(*******************************************************************************
                          protoc-gen-twincat V0.0.0.0                           
             https://github.bhs-world.com/CorrML/protoc-gen-twincat             
*******************************************************************************)
{attribute 'no_explicit_call' := 'do not call this POU directly'}
{attribute 'no-analysis'}
FUNCTION_BLOCK INTERNAL FINAL FB_Baz IMPLEMENTS I_Message
VAR
    _fbMessageParser : FB_MessageParser(ipMessage:= THIS^);
    _fbMessageWriter : FB_MessageWriter(ipMessage:= THIS^);
    _stBaz : ST_Baz;
    END_VAR

PROPERTY PUBLIC Baz : ST_Baz
GET
Baz := _stBaz;
END_GET
SET
_stBaz := Baz;
END_SET
END_PROPERTY

{attribute 'no-analysis'}
(* Calculates the size of this message in Protocol Buffer wire format, in bytes. *)
METHOD CalculateSize : UDINT
VAR
    nSize : UDINT;
    nRepeatedFieldSize : UDINT;
END_VAR
// fixed32 value = 1;
nSize := nSize + 1 + F_ComputeFixed32Size(nValue:= _stBaz.value);
// string name = 2;
nSize := nSize + 1 + F_ComputeStringSize(anyString:= _stBaz.name);
CalculateSize := nSize;
END_METHOD

(* Merges the data from the specified coded input stream with the current message.*)
METHOD MergeFrom : HRESULT
VAR_IN_OUT
    fbParseCtx : FB_ParseContext;
END_VAR
VAR
    nTag : UDINT;
END_VAR
REPEAT
MergeFrom := fbParseCtx.ReadTag(nTag=> nTag);
IF SUCCEEDED(MergeFrom) AND nTag = 0 THEN
    EXIT;
END_IF;

IF FAILED(MergeFrom) THEN
    RETURN;
END_IF

CASE nTag OF
    16#0D:    // fixed32 value = 1;
        MergeFrom := fbParseCtx.ReadFixed32(nValue=> _stBaz.value); 
    16#12:    // string name = 2;
        MergeFrom := fbParseCtx.ReadString(anyStringOut:= _stBaz.name); 
ELSE
    MergeFrom := fbParseCtx.SkipLastField();
END_CASE

UNTIL (FAILED(MergeFrom) OR nTag = 0)
END_REPEAT
END_METHOD

PROPERTY PUBLIC MessageValue : T_Any
GET
MessageValue := F_ToAnyType(anyArg:= _stBaz);
END_GET
END_PROPERTY

PROPERTY PUBLIC Parser : REFERENCE TO FB_MessageParser
GET
Parser REF= THIS^._fbMessageParser;
END_GET
END_PROPERTY

(* Writer for this message.*)
PROPERTY PUBLIC Writer : REFERENCE TO FB_MessageWriter
GET
Writer REF= THIS^._fbMessageWriter;
END_GET
END_PROPERTY

(* Writes the data to the given coded output stream.*)
METHOD WriteTo : HRESULT
VAR_IN_OUT
	(* Coded output stream to write the data to. *)
	fbWriteCtx	: FB_WriteContext;
END_VAR
// fixed32 value = 1;
WriteTo := fbWriteCtx.WriteTag(1, E_WireType.Fixed32);
IF FAILED(WriteTo) THEN
    RETURN;
END_IF
WriteTo := fbWriteCtx.WriteFixed32(nValue:= _stBaz.value);
IF FAILED(WriteTo) THEN
    RETURN;
END_IF
// string name = 2;
WriteTo := fbWriteCtx.WriteTag(2, E_WireType.LengthDelimited);
IF FAILED(WriteTo) THEN
    RETURN;
END_IF
WriteTo := fbWriteCtx.WriteString(sStringToWrite:= _stBaz.name);
IF FAILED(WriteTo) THEN
    RETURN;
END_IF
END_METHOD

END_FUNCTION_BLOCK

(* stored: Version 1.1.0.1
   POU FB_Baz: Id {55a2305c-18b3-4d91-8353-6df28ca708a6}, SpecialFunc None
   Property Baz: Id {d3e69122-e4dc-4b35-9f19-0eafbe88660d}
   Get Get: Id {db605ff9-67d1-4d19-af81-fffdc6f41174}
   Set Set: Id {b2337fb8-821a-46da-b907-b74b3c5b6a68}
   Method CalculateSize: Id {afac9157-31e5-4be8-8fdc-c4827dadc76f}
   Method MergeFrom: Id {da9f284a-7851-4677-aaff-d150e7b1f602}
   Property MessageValue: Id {a88b944c-8687-4082-8e27-e46db6cef87a}
   Get Get: Id {8761bca3-c117-42a4-81d4-9760208f5f5e}
   Property Parser: Id {726f230f-17bb-4357-97f0-5f09e91105b8}
   Get Get: Id {7c805ceb-3139-4da1-98b3-b9dd2361e523}
   Property Writer: Id {ce365ca8-bc36-4ae0-8027-77c18abc34ee}
   Get Get: Id {ba9d19dc-e466-45bb-a257-ee689183a96a}
   Method WriteTo: Id {9085540f-0373-4271-999a-9fedaffab2e4} *)
